{attribute 'qualified_only'}
{attribute 'strict'}
{attribute 'to_string'}
TYPE MasterStateType :
(
	WAITING := 0, 
	CALIBRATION := 1, 
	ACTIVE := 2,
	TRACKING := 3, 
	ERROR := -1
)SINT := WAITING;
END_TYPE

(* stored: Version 1.1.0.1, ProductVersion 3.1.4024.12
   DUT MasterStateType: Id {926d60d7-66b4-4c29-8b79-ca1f1a695b04} *)
